FUNCTION_BLOCK FB_Block IMPLEMENTS I_Interface
VAR_INPUT
END_VAR
VAR_OUTPUT
END_VAR
VAR
	StrValue : string;
	Data : ST_StandardTypes;
END_VAR

END_FUNCTION_BLOCK

(* stored: Version 1.1.0.1, ProductVersion 3.1.4024.12
   POU FB_Block: Id {12fb5738-f1e6-4453-a55d-59197e24ab5a}, SpecialFunc None *)
